PROGRAM MAIN
VAR
	myDB	: DBAdaptor;
	fbTon 	: TON;
	fbTrig	: R_TRIG;
	SQL : STRING(255) := 'INSERT INTO messagelog (message,timestamp) VALUES($'Interval Triggered$',datetime($'now$'))';
	Debug : DB_FunctionResult;
END_VAR

ACT_Interval();
myDB.udiDatabase_ID := 1;
myDB.TimeOut := T#5S;
IF fbTrig.Q THEN
	Debug := myDB.SQL_Insert(SQL);
END_IF

ACTION ACT_Interval:
fbTon(IN:= NOT fbTon.Q, PT:= T#1S );
fbTrig(CLK:= fbTon.Q);
END_ACTION

END_PROGRAM

(* stored: Version 1.1.0.1, ProductVersion 3.1.0.36
   POU MAIN: Id {778f565f-d71e-412b-bdc8-4a36133276c4}, SpecialFunc None
   Action ACT_Interval: Id {6943b751-c915-48dd-a315-1b312ef568bc} *)
